Staubli VAL3: START.PGX

program start()
begin


end
